FUNCTION_BLOCK AL_TO_AULI (* Composite FB for converting AL (LWORD) adapter to AULI (ULINT) adapter — bit-reinterpretation, value-preserving (destination is same width or wider than the source bit-string). *)
  (* Standard: 61499-2; Description: Copyright (c) 2026 HR Agrartechnik GmbH This program and the accompanying materials are made available under the terms of the Eclipse Public License 2.0 which is available at https://www.eclipse.org/legal/epl-2.0/ SPDX-License-Identifier: EPL-2.0 *)
  (* Version 1.0, 2026-02-17, Franz Höpfinger, HR Agrartechnik GmbH *)
  PACKAGE adapter::conversion::unidirectional;
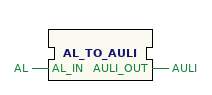
  SOCKETS
    AL_IN : adapter::types::unidirectional::AL; (* LWORD Adapter Input *)
  END_SOCKETS
  PLUGS
    AULI_OUT : adapter::types::unidirectional::AULI; (* ULINT Adapter Output *)
  END_PLUGS
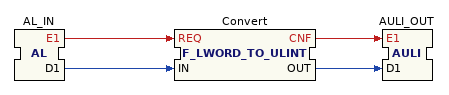
  FBS
    Convert : iec61131::conversion::F_LWORD_TO_ULINT;
  END_FBS
  EVENT_CONNECTIONS
    AL_IN.E1 TO Convert.REQ;
    Convert.CNF TO AULI_OUT.E1;
  END_CONNECTIONS
  DATA_CONNECTIONS
    AL_IN.D1 TO Convert.IN;
    Convert.OUT TO AULI_OUT.D1;
  END_CONNECTIONS
END_FUNCTION_BLOCK
